{attribute 'GeneratedUsingTerminal: EL3751-0000-0020'}
{attribute addProperty BoxType "EL3751-0000-0020"}
{attribute addProperty Id "ARRAY_0DINT4"}
{attribute addProperty CRC "4065202250"}
{attribute addProperty Size "4"}
TYPE Samples_F24E104A :
STRUCT
	{attribute addProperty Name "ARRAY_0"}
	ARRAY_0 : DINT;
END_STRUCT
END_TYPE

(* stored: Version 1.2.0.0, ProductVersion 3.1.4024.9
   DUT Samples_F24E104A: Id {8dfa21a0-606f-463f-8078-953bfa7de75a} *)
